FUNCTION_BLOCK FB_MockTank
VAR_INPUT
	bEnable: BOOL;
	bPumpOn: BOOL;
	rPumpFillRate: REAL:= 50; //litres per second
	rCapacity: REAL:= 500; //litres
	nLowLevelSensorPos: REAL:= 0.2*rCapacity; //percent
	nHighLevelSensorPos: REAL:= 0.8*rCapacity; //percent
	tSamplingRate: TIME:= T#100MS;
END_VAR
VAR_OUTPUT
	rVolume: REAL;
	rConsumption: REAL;
	bLowLevel: BOOL;
	bHighLevel: BOOL;
END_VAR
VAR
	tonConsumptionPeriod: TON;
	rFillRate: REAL;
	fbRandom: DRAND;
	tonSamplingRate: TON;
	rFillRateFactor: REAL;
END_VAR

VAR CONSTANT
	
END_VAR

bLowLevel:= rVolume > nLowLevelSensorPos;
bHighLevel:= rVolume > nHighLevelSensorPos;

tonConsumptionPeriod(IN:= bEnable AND NOT tonConsumptionPeriod.Q, PT:= , Q=> , ET=> );
tonSamplingRate(IN:= NOT tonSamplingRate.Q, PT:= tSamplingRate, Q=> , ET=> );

IF bPumpOn THEN
	rFillRate:= rPumpFillRate;
ELSE
	rFillRate:= 0.0;
END_IF
rFillRateFactor:= TIME_TO_REAL(tonSamplingRate.PT)/1000;

IF bEnable THEN
	IF tonConsumptionPeriod.Q THEN
		fbRandom(seed:=LREAL_TO_INT(fbRandom.Num));
		IF rConsumption = 0.0 THEN
			rConsumption:= LREAL_TO_REAL(fbRandom.Num*rPumpFillRate/2);
			tonConsumptionPeriod.PT:= LREAL_TO_TIME(fbRandom.Num*10000);
		ELSE
			rConsumption:= 0.0;
			tonConsumptionPeriod.PT:= LREAL_TO_TIME(fbRandom.Num*2000);
		END_IF
	END_IF
ELSE
	rConsumption:= 0.0;
END_IF

IF rVolume < 0.0 THEN
	rVolume:= 0.0;
	rConsumption:= 0.0;
END_IF
IF tonSamplingRate.Q THEN
	rVolume:= rVolume + (rFillRate - rConsumption)*rFillRateFactor;
END_IF

END_FUNCTION_BLOCK

(* stored: Version 1.1.0.1, ProductVersion 3.1.4024.12
   POU FB_MockTank: Id {a5d3192f-68c4-4c2c-b9b6-61ff8b767503}, SpecialFunc None *)
